INTERFACE I_SafetyReset EXTENDS I_Cyclic, I_TaskResult

METHOD Execute
VAR_INPUT
END_VAR
END_METHOD

PROPERTY PulseDuration : TIME
SET
END_SET
END_PROPERTY

END_INTERFACE

(* stored: Version 1.1.0.1, ProductVersion 3.1.4026.18
   Itf I_SafetyReset: Id {a612b79d-f306-0613-09d3-a0c4a88a34df}
   Method Execute: Id {21d8f55e-7780-0461-1032-0df0931d5389}
   Property PulseDuration: Id {2601110d-2d60-0d2d-16e5-23efbcee66d8}
   Set Set: Id {f48fed6a-3775-0ceb-020d-ba08c5d8aabe} *)
